Staubli VAL3: start.pgx

program start()
begin
  //call OnStart(tTool,trOffSetOut)
  call OnStart(flange,trOffSetOut)
end
